(* IEC 61131-3 sources: ThesisGitHub/OpenPLC script an ting, 2 files *)

(* ---- A to B conveyor.st ---- *)
PROGRAM program0
  VAR
    I_Sensor AT %IX0.0 : BOOL;
    Q_Conveyor AT %QX0.0 : BOOL;
  END_VAR

  Q_Conveyor := I_Sensor;
END_PROGRAM

CONFIGURATION Config0

  RESOURCE Res0 ON PLC
    TASK task0(INTERVAL := T#20ms,PRIORITY := 0);
    PROGRAM instance0 WITH task0 : program0;
  END_RESOURCE
END_CONFIGURATION

(* ---- FactoryIO Start Stop.st ---- *)
TYPE
  datatype0 : BOOL;
END_TYPE

PROGRAM FactoryIOtest
  VAR
    I_Start AT %IX100.0 : BOOL;
    I_Stop AT %IX100.1 : BOOL;
    Q_Conveyor AT %QX100.0 : BOOL;
  END_VAR

  Q_Conveyor := I_Stop AND (I_Start OR Q_Conveyor);
END_PROGRAM

CONFIGURATION Config0

  RESOURCE Res0 ON PLC
    TASK task0(INTERVAL := T#20ms,PRIORITY := 0);
    PROGRAM instance0 WITH task0 : FactoryIOtest;
  END_RESOURCE
END_CONFIGURATION
